(*	Change the type depending on the needs, minimum packml set or full
Tc3_PackML_V2.ST_PackMLv30 // Tc3_PackML_V2.ST_PackMLv30min*)
TYPE T_PackMLTags : Tc3_PackML_V2.ST_PackMLv30; END_TYPE

(* stored: Version 1.1.0.1, ProductVersion 3.1.4024.9
   DUT T_PackMLTags: Id {1ed0eb96-7045-4fb1-ad91-8e920b725e44} *)
